FUNCTION_BLOCK FB_Station EXTENDS FB_AbstructAsset
VAR_INPUT
END_VAR
VAR_OUTPUT
END_VAR
VAR
	
END_VAR

PROPERTY positioning_job : I_Job
GET
END_GET
SET
END_SET
END_PROPERTY

END_FUNCTION_BLOCK

(* stored: Version 1.1.0.1, ProductVersion 3.1.4026.13
   POU FB_Station: Id {aad04d2c-7b74-4a95-83e2-dc5f6cdfb64a}, SpecialFunc None
   Property positioning_job: Id {0126d3de-6766-4f74-99cf-6d2c3fff12bb}
   Get Get: Id {d4f1fce4-5a26-4b17-85d5-06a2a040cccf}
   Set Set: Id {c2a6e322-7b42-46c4-b1fa-5743e79895b0} *)
